// TIA Portal V20 export
VAR_GLOBAL   // PLC tag table "默认变量表"
END_VAR
